TYPE ST_HOUR_COUNTERS :
STRUCT
	
	TotalHours		: LTIME;
	
	WorkingHours	: LTIME;
END_STRUCT
END_TYPE

(* stored: Version 1.1.0.1, ProductVersion 3.1.4022.11
   DUT ST_HOUR_COUNTERS: Id {8b8e4a80-bd2e-4d39-8e59-97cb0542b2c6} *)
